KUKA KRL data list: mixsort_pick01.dat

&ACCESS RVEO
&REL 49
&COMMENT Sorting station
&PARAM EDITMASK = *
&PARAM DISKPATH = KRC:\R1\Program\MixSortMain
DEFDAT  MIXSORT_PICK01
;***********************************************************
;
; Copyright 2018 - 2025 speedbot All Rights reserved.
;
; File Name: mixsort_pick01.DAT
;
; Description:
;   Language             ==   Krl for KUKA ROBOT
;   Date                 ==   2022 - 06 - 27
;   Modification Data    ==   2025 - 02 - 10
;
; Author: speedbot
;
; Version: 1.1
;***********************************************************

;FOLD EXTERNAL DECLARATIONS;%{PE}%MKUKATPBASIS,%CEXT,%VCOMMON,%P
;FOLD BASISTECH EXT;%{PE}%MKUKATPBASIS,%CEXT,%VEXT,%P
EXT  BAS (BAS_COMMAND  :IN,REAL  :IN )
DECL INT SUCCESS
;ENDFOLD (BASISTECH EXT)
;FOLD USER EXT;%{E}%MKUKATPUSER,%CEXT,%VEXT,%P
;Make your modifications here

;ENDFOLD (USER EXT)
;ENDFOLD (EXTERNAL DECLARATIONS)
DECL MODULEPARAM_T LAST_TP_PARAMS={PARAMS[] "Kuka.VelocityFieldEnabled=True; Kuka.ColDetectFieldEnabled=True; Kuka.MovementParameterFieldEnabled=True; Kuka.IsAngleEnabled=False; Kuka.PointName=P2; Kuka.FrameData.base_no=0; Kuka.FrameData.tool_no=1; Kuka.FrameData.ipo_frame=#BASE; Kuka.isglobalpoint=False; Kuka.MoveDataName=CPDAT4; Kuka.MovementData.cb={AUX_PT {ORI #CONSIDER,E1 #CONSIDER,E2 #CONSIDER,E3 #CONSIDER,E4 #CONSIDER,E5 #CONSIDER,E6 #CONSIDER},TARGET_PT {ORI #INTERPOLATE,E1 #INTERPOLATE,E2 #INTERPOLATE,E3 #INTERPOLATE,E4 #INTERPOLATE,E5 #INTERPOLATE,E6 #INTERPOLATE}}; Kuka.MovementData.apo_fac=50; Kuka.MovementData.apo_dist=100; Kuka.MovementData.axis_acc=100; Kuka.MovementData.axis_vel=100; Kuka.MovementData.circ_typ=#BASE; Kuka.MovementData.jerk_fac=50; Kuka.MovementData.ori_typ=#VAR; Kuka.MovementData.vel=100; Kuka.MovementData.acc=100; Kuka.MovementData.exax_ign=0; Kuka.VelocityPath=0.8; Kuka.BlendingEnabled=False; Kuka.APXEnabled=False; Kuka.CurrentCDSetIndex=0; Kuka.MoveDataPtpName=PDAT3; Kuka.MovementDataPdat.apo_mode=#CDIS; Kuka.MovementDataPdat.apo_dist=500; Kuka.VelocityPtp=100; Kuka.FrameData.point2=; Kuka.MovementData.gear_jerk=100; BASIC.FRAMENAME=OffsRUp; BASIC.X_=0; BASIC.Y_=0; BASIC.Z_=200; BASIC.A_=0; BASIC.B_=0; BASIC.C_=0; BASIC.SOURCENAME=PickPos; BASIC.OFFSFRAME=OffsRUp; BASIC.OFFSETNAME=PickPosRUp; PLC.SEGMENTID=23; PLC.MAGTOOLCTRLMODE=#ON; PLC.TIMEOUT=0; PLC.SLEEPTIME=500; PLC.SUCCESS=Success1  "}
DECL E6POS XPickPos={X 1765.00,Y 0.0,Z 1784.00,A 0.0,B 90.0000,C 0.0,S 2,T 2,E1 0.0,E2 0.0,E3 0.0,E4 0.0,E5 0.0,E6 0.0}
DECL FDAT FPickPos={TOOL_NO 1,BASE_NO 0,IPO_FRAME #BASE,POINT2[] " "}
DECL LDAT LCPDAT2={VEL 0.600000,ACC 100.000,APO_DIST 500.000,APO_FAC 50.0000,AXIS_VEL 100.000,AXIS_ACC 100.000,ORI_TYP #VAR,CIRC_TYP #BASE,JERK_FAC 50.0000,GEAR_JERK 100.000,EXAX_IGN 0}
DECL E6POS XPickPosUp={X 0.0,Y 0.0,Z 0.0,A 0.0,B 0.0,C 0.0,S 0,T 0,E1 0.0,E2 0.0,E3 0.0,E4 0.0,E5 0.0,E6 0.0}
DECL FDAT FPickPosUp={TOOL_NO 1,BASE_NO 0,IPO_FRAME #BASE,POINT2[] " "}
DECL LDAT LCPDAT3={VEL 1.50000,ACC 100.000,APO_DIST 100.000,APO_FAC 50.0000,AXIS_VEL 100.000,AXIS_ACC 100.000,ORI_TYP #VAR,CIRC_TYP #BASE,JERK_FAC 50.0000,GEAR_JERK 100.000,EXAX_IGN 0}
DECL E6POS XPickPosRUp={X 0.0,Y 0.0,Z 0.0,A 0.0,B 0.0,C 0.0,S 0,T 0,E1 0.0,E2 0.0,E3 0.0,E4 0.0,E5 0.0,E6 0.0}
DECL FDAT FPickPosRUp={TOOL_NO 1,BASE_NO 0,IPO_FRAME #BASE,POINT2[] " "}
DECL LDAT LCPDAT4={VEL 0.800000,ACC 100.000,APO_DIST 100.000,APO_FAC 50.0000,AXIS_VEL 100.000,AXIS_ACC 100.000,ORI_TYP #VAR,CIRC_TYP #BASE,JERK_FAC 50.0000,GEAR_JERK 100.000,EXAX_IGN 0}
DECL E6POS XP1={X 1765.00,Y 0.0,Z 1784.00,A 0.0,B 90.0000,C 0.0,S 2,T 2,E1 0.0,E2 0.0,E3 0.0,E4 0.0,E5 0.0,E6 0.0}
DECL FDAT FP1={TOOL_NO 1,BASE_NO 0,IPO_FRAME #BASE,POINT2[] " "}
DECL PDAT PPDAT2={VEL 100.000,ACC 100.000,APO_DIST 500.000,APO_MODE #CDIS,GEAR_JERK 100.000,EXAX_IGN 0}
DECL E6POS XP2={X 1765.00,Y 0.0,Z 1784.00,A 0.0,B 90.0000,C 0.0,S 2,T 2,E1 0.0,E2 0.0,E3 0.0,E4 0.0,E5 0.0,E6 0.0}
DECL FDAT FP2={TOOL_NO 1,BASE_NO 0,IPO_FRAME #BASE,POINT2[] " "}
DECL PDAT PPDAT3={VEL 100.000,ACC 100.000,APO_DIST 500.000,APO_MODE #CDIS,GEAR_JERK 100.000,EXAX_IGN 0}
DECL FRAME OffsUp={X 0.0,Y 0.0,Z 0.0,A 0.0,B 0.0,C 0.0}
DECL FRAME OffsRUp={X 0.0,Y 0.0,Z 0.0,A 0.0,B 0.0,C 0.0}
DECL part_data_t CopyPartData
DECL BOOL Success1 = FALSE
DECL INT PickRetryCount=1
ENDDAT
